(* IEC 61131-3 sources: pandora/pandora/aws-platform-main/aws-platform-main/test/Mocks/Motion, 5 files *)

(* ---- AnalogAxisMock.st ---- *)
USING Esab.Utils.Assets.Mock;
USING Esab.Mock;
USING Esab.Utils.Assets;
USING Esab.Motion;

NAMESPACE Esab.Motion.Mock

    CLASS AnalogAxisMock EXTENDS Asset IMPLEMENTS IAxis
        VAR PUBLIC
            InvalidateHomingMock : MethodMock;
            SetObjectRadiusMock : LRealMethodMock;
            SetJogSpeedMock : LRealMethodMock;
            SetJogHighSpeedMock : LRealMethodMock;
            GetObjectRadiusMock : LRealMethodMock;
            GetObjectCircumferenceMock : LRealMethodMock;
            GetObjectPositionMock : LRealMethodMock;
            GetJogSpeedMock : LRealMethodMock;
            GetJogHighSpeedMock : LRealMethodMock;
            PowerOnMock : MethodMock;
            PowerOffMock : MethodMock;
            ResetMock : BoolMethodMock;
            ExecutePositioningCommandMock : Esab.Motion.Mock.ExecutePositioningCommandMethodMock;
            ExecutePositioningCommandModeMock : ExecutePositioningCommandMethodMock;
            ExecuteHomingCommandMock : Esab.Motion.Mock.ExecuteHomingCommandMethodMock;
            HaltMock : MethodMock;
            JogPositiveMock : BoolMethodMock;
            JogNegativeMock : BoolMethodMock;
            IsEnabledMock : BoolMethodMock;
            IsBusyMock : BoolMethodMock;
            HasErrorMock : BoolMethodMock;
            AtStandstillMock : BoolMethodMock;
            IsHomedMock : BoolMethodMock;
            ActualLinearPositionMock : LRealMethodMock;
            ActualLinearVelocityMock : LRealMethodMock;
            ActualAngularPositionMock : LRealMethodMock;
            ActualAngularVelocityMock : LRealMethodMock;
        END_VAR

        METHOD PUBLIC MockReset
            InvalidateHomingMock.Reset();
            SetObjectRadiusMock.Reset();
            GetObjectRadiusMock.Reset();
            GetObjectCircumferenceMock.Reset();
            GetObjectPositionMock.Reset();
            PowerOnMock.Reset();
            PowerOffMock.Reset();
            ResetMock.Reset();
            ExecutePositioningCommandMock.Reset();
            ExecuteHomingCommandMock.Reset();
            HaltMock.Reset();
            JogPositiveMock.Reset();
            JogNegativeMock.Reset();
            IsEnabledMock.Reset();
            IsBusyMock.Reset();
            HasErrorMock.Reset();
            AtStandstillMock.Reset();
            IsHomedMock.Reset();
            ActualLinearPositionMock.Reset();
            ActualLinearVelocityMock.Reset();
            ActualAngularPositionMock.Reset();
            ActualAngularVelocityMock.Reset();
        END_METHOD

        METHOD PUBLIC InvalidateHoming
            InvalidateHomingMock.IncrementCallCount();
        END_METHOD

        METHOD PUBLIC SetJogSpeed
            VAR_INPUT
                value : LREAL;
            END_VAR

            SetJogSpeedMock.Value := value;
            SetJogSpeedMock.IncrementCallCount();
        END_METHOD

        METHOD PUBLIC SetJogHighSpeed
            VAR_INPUT
                value : LREAL;
            END_VAR

            SetJogHighSpeedMock.Value := value;
            SetJogHighSpeedMock.IncrementCallCount();
        END_METHOD

        METHOD PUBLIC SetObjectRadius
            VAR_INPUT
                value : LREAL;
            END_VAR

            SetObjectRadiusMock.Value := value;
            SetObjectRadiusMock.IncrementCallCount();
        END_METHOD

        METHOD PUBLIC GetObjectRadius : LREAL
            GetObjectRadius := GetObjectRadiusMock.Value;
            GetObjectRadiusMock.IncrementCallCount();
        END_METHOD

        METHOD PUBLIC GetObjectCircumference : LREAL
            GetObjectCircumference := GetObjectCircumferenceMock.Value;
            GetObjectCircumferenceMock.IncrementCallCount();
        END_METHOD

        METHOD PUBLIC GetObjectPosition : LREAL
            GetObjectPosition := GetObjectPositionMock.Value;
            GetObjectPositionMock.IncrementCallCount();
        END_METHOD

        METHOD PUBLIC GetJogSpeed : LREAL;
            GetJogSpeed := GetJogSpeedMock.Value;
            GetJogSpeedMock.IncrementCallCount();
        END_METHOD

        METHOD PUBLIC GetJogHighSpeed : LREAL;
            GetJogHighSpeed := GetJogHighSpeedMock.Value;
            GetJogHighSpeedMock.IncrementCallCount();
        END_METHOD

        METHOD PUBLIC PowerOn
            PowerOnMock.IncrementCallCount();
        END_METHOD

        METHOD PUBLIC PowerOff
            PowerOffMock.IncrementCallCount();
        END_METHOD

        METHOD PUBLIC Reset
            VAR_INPUT
                Restart : BOOL;
            END_VAR

            ResetMock.Value := Restart;
            ResetMock.IncrementCallCount();
        END_METHOD

        METHOD PUBLIC ExecutePositioningCommand : AxisCommandError
            VAR_INPUT
                command : AxisPositioningCommand;
            END_VAR

            ExecutePositioningCommandMock.Command := command;
            ExecutePositioningCommandMock.IncrementCallCount();
        END_METHOD

        METHOD PUBLIC ExecuteHomingCommand : AxisCommandError
            VAR_INPUT
                command : AxisHomingCommand;
            END_VAR

            ExecuteHomingCommandMock.Command := command;
            ExecuteHomingCommandMock.IncrementCallCount();
        END_METHOD

        METHOD PUBLIC Halt
            HaltMock.IncrementCallCount();
        END_METHOD

        METHOD PUBLIC JogPositive
            VAR_INPUT
                highSpeed : BOOL := FALSE;
            END_VAR

            JogPositiveMock.Value := highSpeed;
            JogPositiveMock.IncrementCallCount();
        END_METHOD

        METHOD PUBLIC JogNegative
            VAR_INPUT
                highSpeed : BOOL := FALSE;
            END_VAR

            JogNegativeMock.Value := highSpeed;
            JogNegativeMock.IncrementCallCount();
        END_METHOD

        METHOD PUBLIC IsEnabled : BOOL
            IsEnabled := IsEnabledMock.Value;
            IsEnabledMock.IncrementCallCount();
        END_METHOD

        METHOD PUBLIC IsBusy : BOOL
            IsBusy := IsBusyMock.Value;
            IsBusyMock.IncrementCallCount();
        END_METHOD

        METHOD PUBLIC HasError : BOOL
            HasError := HasErrorMock.Value;
            HasErrorMock.IncrementCallCount();
        END_METHOD

        METHOD PUBLIC AtStandstill : BOOL
            AtStandstill := AtStandstillMock.Value;
            AtStandstillMock.IncrementCallCount();
        END_METHOD

        METHOD PUBLIC IsHomed : BOOL
            IsHomed := IsHomedMock.Value;
            IsHomedMock.IncrementCallCount();
        END_METHOD

        METHOD PUBLIC ActualLinearPosition : LREAL
            ActualLinearPosition := ActualLinearPositionMock.Value;
            ActualLinearPositionMock.IncrementCallCount();
        END_METHOD

        METHOD PUBLIC ActualLinearVelocity : LREAL
            ActualLinearVelocity := ActualLinearVelocityMock.Value;
            ActualLinearVelocityMock.IncrementCallCount();
        END_METHOD

        METHOD PUBLIC ActualAngularPosition : LREAL
            ActualAngularPosition := ActualAngularPositionMock.Value;
            ActualAngularPositionMock.IncrementCallCount();
        END_METHOD

        METHOD PUBLIC ActualAngularVelocity : LREAL
            ActualAngularVelocity := ActualAngularVelocityMock.Value;
            ActualAngularVelocityMock.IncrementCallCount();
        END_METHOD

        METHOD PUBLIC OVERRIDE Observe : IAssetObservable
            Observe := NULL;
        END_METHOD
    END_CLASS
END_NAMESPACE

(* ---- HighSpeedCounterMock.st ---- *)
USING Esab.Mock;
USING Esab.Io;

NAMESPACE Esab.Io.Mock

    CLASS HighSpeedCounterMock IMPLEMENTS IHighSpeedCounter
        VAR PUBLIC
            ExecuteMock : MethodMock;
            SetHardwareConfigurationMock : HighSpeedCounterHardwareConfigurationMethodMock;
            EnableMock : MethodMock;
            DisableMock : MethodMock;
            GetCountValueMock  : DIntMethodMock;
            GetMeasuredValueMock : DIntMethodMock;
            GetUpperCountingLimitMock : DIntMethodMock;
            GetLowerCountingLimitMock : DIntMethodMock;
            SetCountValueMock : DIntMethodMock;
            HasErrorMock : BoolMethodMock;
            GetErrorIdMock : WordMethodMock;
        END_VAR

        METHOD PUBLIC MockReset
            ExecuteMock.Reset();
            EnableMock.Reset();
            DisableMock.Reset();
            GetCountValueMock.Reset();
            GetMeasuredValueMock.Reset();
            SetCountValueMock.Reset();
            HasErrorMock.Reset();
            GetErrorIdMock.Reset();
        END_METHOD

        METHOD PUBLIC Execute
            ExecuteMock.IncrementCallCount();
        END_METHOD

        METHOD PUBLIC SetHardwareConfiguration
            VAR_INPUT
                hwConfiguration : REF_TO HighSpeedCounterHardwareConfiguration;
            END_VAR

            SetHardwareConfigurationMock.Value := hwConfiguration;
            SetHardwareConfigurationMock.IncrementCallCount();
        END_METHOD

        METHOD PUBLIC Enable
            EnableMock.IncrementCallCount();
        END_METHOD

        METHOD PUBLIC Disable
            DisableMock.IncrementCallCount();
        END_METHOD

        METHOD PUBLIC GetCountValue : DINT
            GetCountValueMock.IncrementCallCount();
            GetCountValue := GetCountValueMock.Value;
        END_METHOD

        METHOD PUBLIC GetMeasuredValue : DINT
            GetMeasuredValueMock.IncrementCallCount();
            GetMeasuredValue := GetMeasuredValueMock.Value;
        END_METHOD

        METHOD PUBLIC GetUpperCountingLimit : DINT
            GetUpperCountingLimitMock.IncrementCallCount();
            GetUpperCountingLimit := GetUpperCountingLimitMock.Value;
        END_METHOD

        METHOD PUBLIC GetLowerCountingLimit : DINT
            GetLowerCountingLimitMock.IncrementCallCount();
            GetLowerCountingLimit := GetLowerCountingLimitMock.Value;
        END_METHOD

        METHOD PUBLIC SetCountValue
            VAR_INPUT
                value : DINT;
            END_VAR

            SetCountValueMock.IncrementCallCount();
            SetCountValueMock.Value := value;
        END_METHOD

        METHOD PUBLIC HasError : BOOL
            HasErrorMock.IncrementCallCount();
            HasError := HasErrorMock.Value;
        END_METHOD

        METHOD PUBLIC GetErrorId : WORD
            GetErrorIdMock.IncrementCallCount();
            GetErrorId := GetErrorIdMock.Value;
        END_METHOD
    END_CLASS

    CLASS HighSpeedCounterHardwareConfigurationMethodMock EXTENDS MethodMock
        VAR PUBLIC
            Value : REF_TO HighSpeedCounterHardwareConfiguration;
        END_VAR

        METHOD PUBLIC OVERRIDE Reset
            Value := NULL;
            SUPER.Reset();
        END_METHOD
    END_CLASS

END_NAMESPACE

(* ---- SpeedWheelMock.st ---- *)
USING Esab.Motion.MeasurementSystem;
USING Esab.Mock;

NAMESPACE Esab.Motion.MeasurementSystems.Mock

    CLASS SpeedWheelMock IMPLEMENTS IMeasurementSystem1D
        VAR PUBLIC
            IsInitializedMock : BoolMethodMock;
            ExecuteMock : MethodMock;
            GetMeasuredPositionMock : LRealMethodMock;
            GetMeasuredVelocityMock : LRealMethodMock;
            ResetMeasuredPositionMock : MethodMock;
            SetListenerMock : MethodMock;
        END_VAR

        METHOD PUBLIC MockReset
            IsInitializedMock.Reset();
            ExecuteMock.Reset();
            GetMeasuredPositionMock.Reset();
            GetMeasuredVelocityMock.Reset();
            ResetMeasuredPositionMock.Reset();
            SetListenerMock.Reset();
        END_METHOD

        METHOD PUBLIC IsInitialized : BOOL
            IsInitializedMock.IncrementCallCount();
            IsInitialized := IsInitializedMock.Value;
        END_METHOD

        METHOD PUBLIC Execute
            ExecuteMock.IncrementCallCount();
        END_METHOD

        METHOD PUBLIC GetMeasuredPosition : LREAL
            GetMeasuredPositionMock.IncrementCallCount();
            GetMeasuredPosition := GetMeasuredPositionMock.Value;
        END_METHOD

        METHOD PUBLIC GetMeasuredVelocity : LREAL
            GetMeasuredVelocityMock.IncrementCallCount();
            GetMeasuredVelocity := GetMeasuredVelocityMock.Value;
        END_METHOD

        METHOD PUBLIC ResetMeasuredPosition
            ResetMeasuredPositionMock.IncrementCallCount();
        END_METHOD

        METHOD PUBLIC SetListener
            VAR_INPUT
                listener : IMeasurementSystemListener;
            END_VAR

            SetListenerMock.IncrementCallCount();
        END_METHOD
    END_CLASS

END_NAMESPACE

(* ---- ToPosAxisMock.st ---- *)
USING Esab.Mock;
USING Esab.Utils.Assets;

NAMESPACE Esab.Motion.Mock

    CLASS ToPosAxisMock EXTENDS Asset IMPLEMENTS IAxis
        VAR PUBLIC
            PowerOnMock : MethodMock;
            PowerOffMock : MethodMock;
            ResetMock : MethodMock;
            ExecuteMock : MethodMock;
            ExecutePositioningCommandMock : ExecutePositioningCommandMethodMock;
            ExecuteHomingCommandMock : ExecuteHomingCommandMethodMock;
            InvalidateHomingMock : MethodMock;
            HaltMock : MethodMock;
            SetJogSpeedMock : LRealMethodMock;
            SetJogHighSpeedMock : LRealMethodMock;
            SetObjectRadiusMock : LRealMethodMock;
            JogPositiveMock : BoolMethodMock;
            JogNegativeMock : BoolMethodMock;
            IsEnabledMock : BoolMethodMock;
            IsBusyMock : BoolMethodMock;
            HasErrorMock : BoolMethodMock;
            AtStandstillMock : BoolMethodMock;
            IsHomedMock : BoolMethodMock;
            ActualLinearPositionMock : LRealMethodMock;
            ActualLinearVelocityMock : LRealMethodMock;
            ActualAngularPositionMock : LRealMethodMock;
            ActualAngularVelocityMock : LRealMethodMock;
        END_VAR

        VAR PRIVATE
            _observable : AxisObservable;
        END_VAR

        METHOD PUBLIC MockReset
            PowerOnMock.Reset();
            PowerOffMock.Reset();
            ResetMock.Reset();
            ExecuteMock.Reset();
            ExecutePositioningCommandMock.Reset();
            ExecuteHomingCommandMock.Reset();
            HaltMock.Reset();
            IsEnabledMock.Reset();
            IsBusyMock.Reset();
            HasErrorMock.Reset();
            AtStandstillMock.Reset();
            IsHomedMock.Reset();
            ActualLinearPositionMock.Reset();
            ActualLinearVelocityMock.Reset();
            ActualAngularPositionMock.Reset();
            ActualAngularVelocityMock.Reset();
        END_METHOD

        METHOD PUBLIC PowerOn
            PowerOnMock.IncrementCallCount();
        END_METHOD

        METHOD PUBLIC PowerOff
            PowerOffMock.IncrementCallCount();
        END_METHOD

        METHOD PUBLIC Reset
            VAR_INPUT
                Restart : BOOL;
            END_VAR

            ResetMock.IncrementCallCount();
        END_METHOD

        METHOD PUBLIC OVERRIDE Execute
            ExecuteMock.IncrementCallCount();
        END_METHOD

        METHOD PUBLIC ExecutePositioningCommand : AxisCommandError
            VAR_INPUT
                command: AxisPositioningCommand;
            END_VAR

            ExecutePositioningCommandMock.IncrementCallCount();
            ExecutePositioningCommandMock.Command := command;
        END_METHOD

        METHOD PUBLIC ExecuteHomingCommand : AxisCommandError
            VAR_INPUT
                command: AxisHomingCommand;
            END_VAR

            ExecuteHomingCommandMock.IncrementCallCount();
            ExecuteHomingCommandMock.Command := command;
        END_METHOD

        METHOD PUBLIC InvalidateHoming
            ;
        END_METHOD

        METHOD PUBLIC Halt
            HaltMock.IncrementCallCount();
        END_METHOD

        METHOD PUBLIC SetJogSpeed
            VAR_INPUT
                value : LREAL;
            END_VAR

            SetJogSpeedMock.Value := value;
            SetJogSpeedMock.IncrementCallCount();
        END_METHOD

        METHOD PUBLIC SetJogHighSpeed
            VAR_INPUT
                value : LREAL;
            END_VAR

            SetJogHighSpeedMock.Value := value;
            SetJogHighSpeedMock.IncrementCallCount();
        END_METHOD

        METHOD PUBLIC SetObjectRadius
            VAR_INPUT
                value : LREAL;
            END_VAR

            SetObjectRadiusMock.Value := value;
            SetObjectRadiusMock.IncrementCallCount();
        END_METHOD

        METHOD PUBLIC JogPositive
            VAR_INPUT
                highSpeed : BOOL := FALSE;
            END_VAR

            JogPositiveMock.Value := highSpeed;
            JogPositiveMock.IncrementCallCount();
        END_METHOD

        METHOD PUBLIC JogNegative
            VAR_INPUT
                highSpeed : BOOL := FALSE;
            END_VAR

            JogNegativeMock.Value := highSpeed;
            JogNegativeMock.IncrementCallCount();
        END_METHOD

        METHOD PUBLIC IsEnabled : BOOL
            IsEnabled := IsEnabledMock.Value;
            IsEnabledMock.IncrementCallCount();
        END_METHOD

        METHOD PUBLIC IsBusy : BOOL
            IsBusy := IsBusyMock.Value;
            IsBusyMock.IncrementCallCount();
        END_METHOD

        METHOD PUBLIC HasError : BOOL
            HasError := HasErrorMock.Value;
            HasErrorMock.IncrementCallCount();
        END_METHOD

        METHOD PUBLIC AtStandstill : BOOL
            AtStandstill := AtStandstillMock.Value;
            AtStandstillMock.IncrementCallCount();
        END_METHOD

        METHOD PUBLIC IsHomed : BOOL
            IsHomed := IsHomedMock.Value;
            IsHomedMock.IncrementCallCount();
        END_METHOD

        METHOD PUBLIC ActualLinearPosition : LREAL
            ActualLinearPosition := ActualLinearPositionMock.Value;
            ActualLinearPositionMock.IncrementCallCount();
        END_METHOD

        METHOD PUBLIC ActualLinearVelocity : LREAL
            ActualLinearVelocity := ActualLinearVelocityMock.Value;
            ActualLinearVelocityMock.IncrementCallCount();
        END_METHOD

        METHOD PUBLIC ActualAngularPosition : LREAL
            ActualAngularPosition := ActualAngularPositionMock.Value;
            ActualAngularPositionMock.IncrementCallCount();
        END_METHOD

        METHOD PUBLIC ActualAngularVelocity : LREAL
            ActualAngularVelocity := ActualAngularVelocityMock.Value;
            ActualAngularVelocityMock.IncrementCallCount();
        END_METHOD

        METHOD PUBLIC OVERRIDE Observe : IAssetObservable
            Observe := _observable;
        END_METHOD
    END_CLASS

    CLASS ExecutePositioningCommandMethodMock EXTENDS MethodMock
        VAR PUBLIC
            Command : AxisPositioningCommand;
        END_VAR

        VAR PRIVATE
            _defaultCommand : AxisPositioningCommand;
        END_VAR

        METHOD PUBLIC OVERRIDE Reset
            SUPER.Reset();
            Command := _defaultCommand;
        END_METHOD
    END_CLASS

    CLASS ExecuteHomingCommandMethodMock EXTENDS MethodMock
        VAR PUBLIC
            Command : AxisHomingCommand;
        END_VAR

        VAR PRIVATE
            _defaultCommand : AxisHomingCommand;
        END_VAR

        METHOD PUBLIC OVERRIDE Reset
            SUPER.Reset();
            Command := _defaultCommand;
        END_METHOD
    END_CLASS

END_NAMESPACE

(* ---- WeldHeadManipulator.st ---- *)
USING Esab.Mock;
USING Esab.Utils.Assets;
USING Esab.Mock;

NAMESPACE Esab.Motion.Mock
    CLASS WeldHeadManipulatorMock EXTENDS Asset IMPLEMENTS IWeldHeadManipulator
        VAR PUBLIC
            EnableMock : WeldHeadManipulatorErrorCodeMock;
            DisableMock : MethodMock;
            MoveInterpolatedMock : MoveInterpolatedMethodMock;
            MoveMock : MoveMethodMock;
            IsEnabledMock : BoolMethodMock;
            GetPositionMock : LRealArray2MethodMock;
            GetSpeedMock : LRealMethodMock;
            GetVelocityMock : LRealArray2MethodMock;
            GetControlModeMock : GetControlModeMethodMock;
            SetControlModeMock : SetControlModeMethodMock;
        END_VAR

        METHOD PUBLIC MockReset
            EnableMock.Reset();
            DisableMock.Reset();
            MoveMock.Reset();
            IsEnabledMock.Reset();
            GetPositionMock.Reset();
            GetSpeedMock.Reset();
            GetVelocityMock.Reset();
            GetControlModeMock.Reset();
            SetControlModeMock.Reset();
        END_METHOD

        METHOD PUBLIC Enable : WeldHeadManipulatorErrorCode
            EnableMock.IncrementCallCount();
            Enable := EnableMock.ErrorCode;
        END_METHOD

        METHOD PUBLIC Disable
            DisableMock.IncrementCallCount();
        END_METHOD

        METHOD PUBLIC Move : WeldHeadManipulatorErrorCode
            VAR_INPUT
                position : ARRAY [0..1] OF LREAL := [0.0, 0.0];
                speed : LREAL := -1;
            END_VAR

            MoveInterpolatedMock.Speed := speed;
            MoveInterpolatedMock.Position := position;
            MoveInterpolatedMock.IncrementCallCount();
            Move := MoveMock.ErrorCode;
        END_METHOD

        METHOD PUBLIC Move : WeldHeadManipulatorErrorCode
            VAR_INPUT
                position : ARRAY [0..1] OF LREAL := [0.0, 0.0];
                speed : ARRAY [0..1] OF LREAL := [-1.0, -1.0];
            END_VAR

            MoveMock.Speed := speed;
            MoveMock.Position := position;
            MoveMock.IncrementCallCount();
            Move := MoveMock.ErrorCode;
        END_METHOD

        METHOD PUBLIC IsEnabled : BOOL
            IsEnabledMock.IncrementCallCount();
            IsEnabled := IsEnabledMock.Value;
        END_METHOD

        METHOD PUBLIC OVERRIDE Observe : IAssetObservable
            Observe := NULL;
        END_METHOD

        METHOD PUBLIC GetPosition : ARRAY [0..1] OF LREAL
            GetPositionMock.IncrementCallCount();
            GetPosition := GetPositionMock.Value;
        END_METHOD

        METHOD PUBLIC GetSpeed : LREAL
            GetSpeedMock.IncrementCallCount();
            GetSpeed := GetSpeedMock.Value;
        END_METHOD

        METHOD PUBLIC GetVelocity : ARRAY [0..1] OF LREAL
            GetVelocityMock.IncrementCallCount();
            GetVelocity := GetVelocityMock.Value;
        END_METHOD

        METHOD PUBLIC GetControlMode : WeldHeadManipulatorControlMode
            GetControlModeMock.IncrementCallCount();
            GetControlMode := GetControlModeMock.ControlMode;
        END_METHOD

        METHOD PUBLIC SetControlMode
            VAR_INPUT
                controlMode : WeldHeadManipulatorControlMode;
            END_VAR

            SetControlModeMock.ControlMode := controlMode;
            SetControlModeMock.IncrementCallCount();
        END_METHOD
    END_CLASS

    CLASS MoveInterpolatedMethodMock EXTENDS WeldHeadManipulatorErrorCodeMock
        VAR PUBLIC
            Speed : LREAL;
            Position : ARRAY [0..1] OF LREAL;
        END_VAR

        METHOD PUBLIC OVERRIDE Reset
            SUPER.Reset();

            Speed := -1.0;
            Position[0] := 0.0;
            Position[1] := 0.0;
        END_METHOD
    END_CLASS

    CLASS MoveMethodMock EXTENDS WeldHeadManipulatorErrorCodeMock
        VAR PUBLIC
            Speed : ARRAY [0..1] OF LREAL;
            Position : ARRAY [0..1] OF LREAL;
        END_VAR

        METHOD PUBLIC OVERRIDE Reset
            SUPER.Reset();

            Speed[0] := -1.0;
            Speed[1] := -1.0;
            Position[0] := 0.0;
            Position[1] := 0.0;
        END_METHOD
    END_CLASS

    CLASS GetControlModeMethodMock EXTENDS WeldHeadManipulatorControlModeMock
    END_CLASS

    CLASS SetControlModeMethodMock EXTENDS MethodMock
        VAR PUBLIC
            ControlMode : WeldHeadManipulatorControlMode := WeldHeadManipulatorControlMode#NoControl;
        END_VAR

        METHOD PUBLIC OVERRIDE Reset
            SUPER.Reset();

            ControlMode := WeldHeadManipulatorControlMode#NoControl;
        END_METHOD
    END_CLASS

    CLASS WeldHeadManipulatorErrorCodeMock EXTENDS MethodMock
        VAR PUBLIC
            ErrorCode : WeldHeadManipulatorErrorCode;
        END_VAR

        METHOD PUBLIC OVERRIDE Reset
            SUPER.Reset();

            ErrorCode := WeldHeadManipulatorErrorCode#NoError;
        END_METHOD
    END_CLASS

    CLASS WeldHeadManipulatorControlModeMock EXTENDS MethodMock
        VAR PUBLIC
            ControlMode : WeldHeadManipulatorControlMode;
        END_VAR

        METHOD PUBLIC OVERRIDE Reset
            SUPER.Reset();

            ControlMode := WeldHeadManipulatorControlMode#NoControl;
        END_METHOD
    END_CLASS

    CLASS LRealArray2MethodMock EXTENDS MethodMock
        VAR PUBLIC
            Value : ARRAY [0..1] OF LREAL;
        END_VAR

        METHOD PUBLIC OVERRIDE Reset
            SUPER.Reset();
            Value[0] := 0.0;
            Value[1] := 0.0;
        END_METHOD
    END_CLASS
END_NAMESPACE
